(* Logix 5000 project; controller Close_Palletizing 1769-L33ERM rev 33.13; software revision 33.00; part 5 of 5 *)
(* tags used below, declared in another part *)
   ConveyorLocations_ONS : BOOL;
   Write_ActiveUserFrame2 : BOOL;
   ActiveUserFrame : DINT;
   ActiveUserFrame_Old : DINT;
   ActiveUserFrame_Timer : TIMER;
   ActiveUserFrameErr : BOOL;
   AirPressure : ALIAS FOR YRC1000_Rbt_Ctlr:I.Data[1].4;   // Sensor on air in, used to verify pressure
   BoltBucketSensor : ALIAS FOR YRC1000_Rbt_Ctlr:I.Data[1].7;   // Sense if the Bolt Bucket is present in the stand
   CenterDist : DINT;
   ConveyorApproachLocation : YRC1000_POSITION_VAR;
   ConveyorHeight : REAL;   // Distance from UF 3 to the top of the conveyor
   ConveyorPickLocation : YRC1000_POSITION_VAR;
   CurrentPos : REAL[6];   // Current position of the active TCP on the robot
   CurrentPos_micro : YRC1000_POSITION_VAR;   // μm
   currentPosErr : BOOL;
   CurrPos_Timer : TIMER;
   DoorRequestAccess : ALIAS FOR YRC1000_Rbt_Ctlr:I.Data[1].0;   // Door Interlock, For request Entry
   DoorUnlocked : ALIAS FOR YRC1000_Rbt_Ctlr:I.Data[2].0;   // The Door Latch is unlocked
   Error_RobotPickupFailed : ALIAS FOR YRC1000_Rbt_Ctlr:I.Data[9].3;
   GoToPartChange : ALIAS FOR YRC1000_Rbt_Ctlr:O.Data[6].0;
   HMI_Reset : BOOL;
   HMI_Stop : ALIAS FOR YRC1000_Rbt_Ctlr:O.Data[5].4;
   IFM_Port1_Stroke : Generic_4PORT_IOL;   // Stroke sensor reading can be found in StrokeInputArray[0]
   InPartChange : ALIAS FOR YRC1000_Rbt_Ctlr:I.Data[9].7;
   LayerNum : DINT;
   LeftPalletComplete : ALIAS FOR YRC1000_Rbt_Ctlr:O.Data[4].0;
   LeftPalletPresent : ALIAS FOR YRC1000_Rbt_Ctlr:O.Data[6].6;
   LeftPalletSensor : ALIAS FOR YRC1000_Rbt_Ctlr:I.Data[1].2;   // Sense if a pallet is in the pallet holder
   LeftPalletWillBeNew : BOOL;
   msg_Read_ActiveUserFrame : MESSAGE;
   msg_Read_CurrentPosition : MESSAGE;   // Reading the current position of the robot
   msg_Read_PalletCount : MESSAGE;
   msg_Read_PartCount : MESSAGE;   // Reading Part Count from the robot
   msg_Write_ActiveUserFrame : MESSAGE;
   msg_Write_ConveyorApproachLocation : MESSAGE;
   msg_Write_ConveyorPickLocation : MESSAGE;
   msg_Write_PalletCount : MESSAGE;
   msg_Write_PalletPlaceLocation : MESSAGE;
   msg_Write_PartCount : MESSAGE;
   msg_Write_RadiatorType : MESSAGE;
   OffsetDist : DINT;
   PalletCount : DINT;
   PalletCount_old : DINT;
   PalletCount_Timer : TIMER;
   PalletCountErr : BOOL;
   Palletizer_full_produced : DINT;
   PalletNotClear : ALIAS FOR YRC1000_Rbt_Ctlr:O.Data[6].5;
   PartCount : DINT;
   PartCount_Timer : TIMER;
   PartCountErr : BOOL;
   PartInTool : ALIAS FOR YRC1000_Rbt_Ctlr:O.Data[4].2;
   PartLength : DINT;
   PartLength_Current : DINT;   // 17" = 432 mm | 30" = 762 mm | 41" = 1041 mm
   PartNum : DINT;
   PartNum_Current : DINT;
   PartNumber : STRING;
   PartNumber_Current : STRING;
   PartPosition : DINT;
   PartRows : DINT;
   PartRows_Current : DINT;
   PartThickness : REAL;
   PartThickness_Current : REAL;   // 2r = 34.1-34.6 mm | 3r = 51.1-51.8 mm | 4r = 68.2-68.9 mm
   PartWidth : DINT;
   PartWidth_Current : DINT;   // 14" = 356 mm | 16" = 407 mm | 20" = 508 mm | 22" = 559 mm | 24" = 610 mm | 28" = 711 mm | 32" = 813 mm
   PickReq_State : DINT;
   PickRequest : ALIAS FOR YRC1000_Rbt_Ctlr:I.Data[9].6;
   PickRequestAcknowledge : ALIAS FOR YRC1000_Rbt_Ctlr:O.Data[5].5;
   PickupConveyorSensor : ALIAS FOR YRC1000_Rbt_Ctlr:I.Data[1].5;   // Sense if the radiator is ready for pickup
   Place_Error : BOOL;
   PlaceReq_State : DINT;
   PlaceRequestAcknowledge : ALIAS FOR YRC1000_Rbt_Ctlr:O.Data[4].5;
   PN_Timer : TIMER;
   QuadStack : ALIAS FOR YRC1000_Rbt_Ctlr:O.Data[5].1;
   RadiatorPlaceLocation : YRC1000_POSITION_VAR;
   RadiatorType : DINT;   // 1: 17" 2: 30" 3 41"
   Read_ActiveUserFrame : BOOL;
   Read_CurrPos : BOOL;
   Read_PalletCount : BOOL;
   Read_PartCount : BOOL;
   Reset : ALIAS FOR YRC1000_Rbt_Ctlr:I.Data[1].1;   // Door Interlock, For reset Entry
   ResetPalletCount : BOOL;
   RightPalletComplete : ALIAS FOR YRC1000_Rbt_Ctlr:O.Data[4].1;
   RightPalletPresent : ALIAS FOR YRC1000_Rbt_Ctlr:O.Data[6].7;
   RightPalletSensor : ALIAS FOR YRC1000_Rbt_Ctlr:I.Data[1].3;   // Sense if a pallet is in the pallet holder
   RightPalletWillBeNew : BOOL;
   RobotExternalEStop : ALIAS FOR YRC1000_Rbt_Ctlr:I.Data[4].1;
   RobotPlaceRequest : ALIAS FOR YRC1000_Rbt_Ctlr:I.Data[9].2;
   RobotTeachPendantEStop : ALIAS FOR YRC1000_Rbt_Ctlr:I.Data[4].2;
   Running : ALIAS FOR YRC1000_Rbt_Ctlr:I.Data[8].0;   // Robot running status
   SafetyCircuitBroken : ALIAS FOR YRC1000_Rbt_Ctlr:I.Data[4].0;
   SecondConveyorSensor : ALIAS FOR YRC1000_Rbt_Ctlr:I.Data[1].6;   // Sense if a coil is waiting on the conveyor
   SideDist : DINT;
   SingleStack : ALIAS FOR YRC1000_Rbt_Ctlr:O.Data[5].0;
   test_toggle : BOOL;
   ToolExtended : ALIAS FOR YRC1000_Rbt_Ctlr:O.Data[4].3;
   ToolRetracted : ALIAS FOR YRC1000_Rbt_Ctlr:O.Data[4].4;
   ToPC_AirPressure : DINT;
   ToPC_BoltBucketSensor : DINT;
   ToPC_ConveyorStatus : DINT;
   ToPC_DoorStatus : DINT;
   ToPC_FanucFault : DINT;
   ToPC_FanucRunning : DINT;
   ToPC_LeftPalletStatus : DINT;
   ToPC_PalletNotClear : DINT;
   ToPC_PickupFailed : DINT;
   ToPC_PlaceError : DINT;
   ToPC_RightPalletStatus : DINT;
   ToPC_RobotEStop : DINT;
   ToPC_RobotRunning : DINT;
   ToPC_SafetyCircuitBroken : DINT;
   ToPC_ToolStatus : DINT;
   TwoStack : ALIAS FOR YRC1000_Rbt_Ctlr:O.Data[6].2;
   WaitingForPartAtEnd : BOOL;
   Write_ActiveUserFrame : BOOL;
   Write_ActiveUserFrame1 : BOOL;
   Write_ConveyorLocations : BOOL;
   Write_PalletPlaceLocation : BOOL;
   Write_PartCount : BOOL;
   Write_RadiatorType : BOOL;
(* MainProgram, continued *)

ROUTINE Motoman_Messaging   (* ladder *)
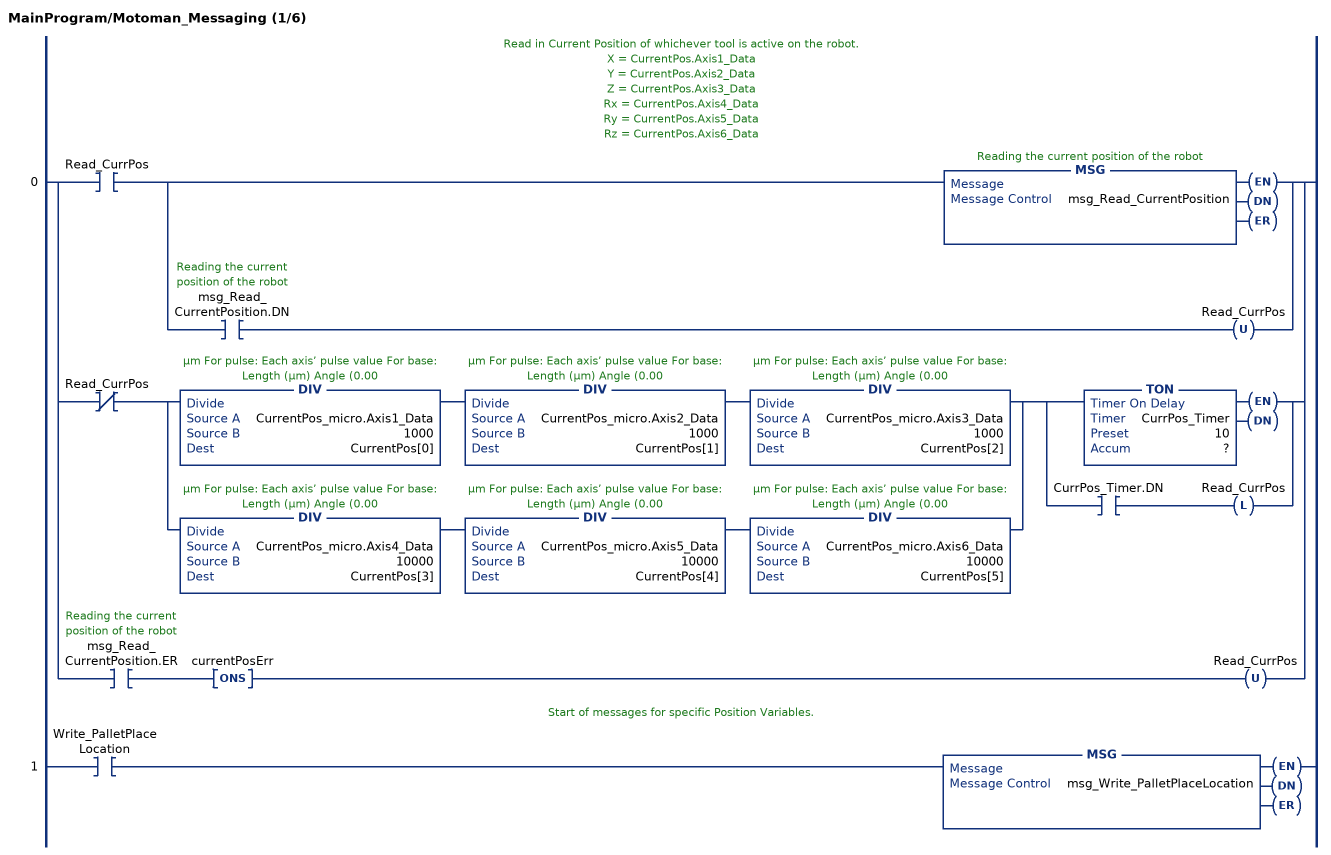
   // Read in Current Position of whichever tool is active on the robot.
   //  X = CurrentPos.Axis1_Data
   //  Y = CurrentPos.Axis2_Data
   //  Z = CurrentPos.Axis3_Data
   // Rx = CurrentPos.Axis4_Data
   // Ry = CurrentPos.Axis5_Data
   // Rz = CurrentPos.Axis6_Data
   0: [XIC(Read_CurrPos) [MSG(msg_Read_CurrentPosition) ,XIC(msg_Read_CurrentPosition.DN) OTU(Read_CurrPos) ] ,XIO(Read_CurrPos) [DIV(CurrentPos_micro.Axis1_Data,1000,CurrentPos[0]) DIV(CurrentPos_micro.Axis2_Data,1000,CurrentPos[1]) DIV(CurrentPos_micro.Axis3_Data,1000,CurrentPos[2]) ,DIV(CurrentPos_micro.Axis4_Data,10000,CurrentPos[3]) DIV(CurrentPos_micro.Axis5_Data,10000,CurrentPos[4]) DIV(CurrentPos_micro.Axis6_Data,10000,CurrentPos[5]) ] [TON(CurrPos_Timer,?,?) ,XIC(CurrPos_Timer.DN) OTL(Read_CurrPos) ] ,XIC(msg_Read_CurrentPosition.ER) ONS(currentPosErr) OTU(Read_CurrPos) ];
   // Start of messages for specific Position Variables.
   1: XIC(Write_PalletPlaceLocation)MSG(msg_Write_PalletPlaceLocation);
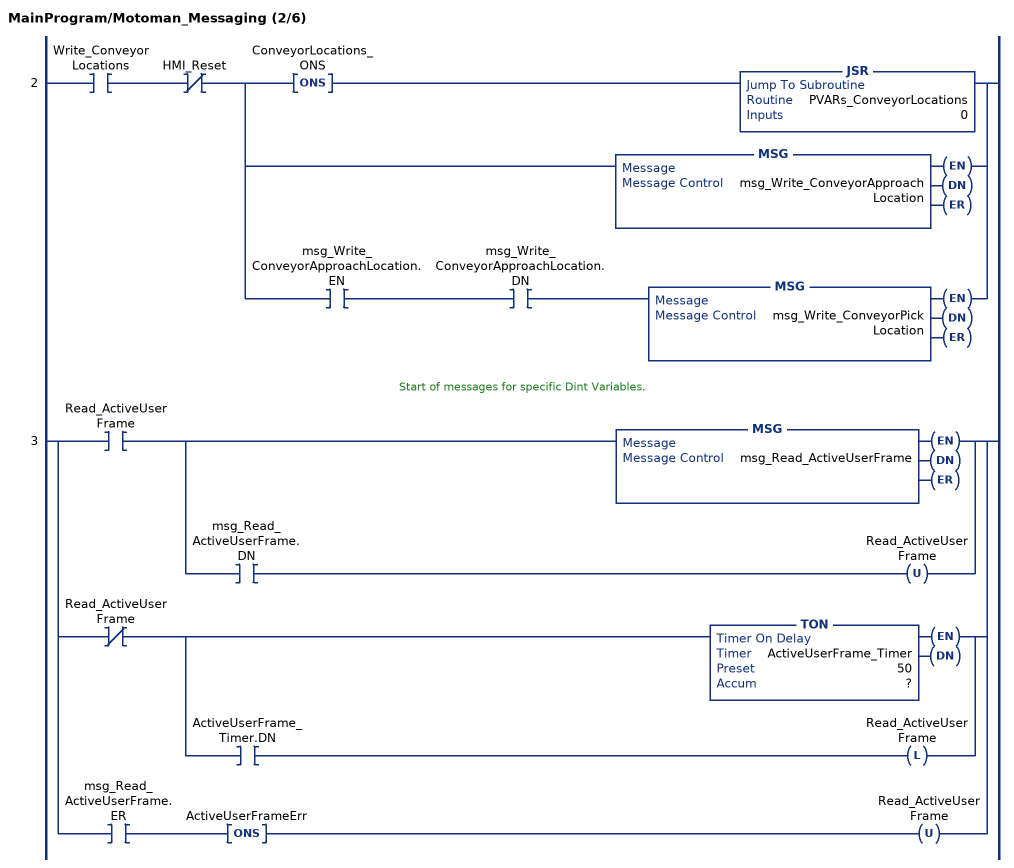
   2: XIC(Write_ConveyorLocations)XIO(HMI_Reset)[ONS(ConveyorLocations_ONS) JSR(PVARs_ConveyorLocations,0) ,MSG(msg_Write_ConveyorApproachLocation) ,XIC(msg_Write_ConveyorApproachLocation.EN) XIC(msg_Write_ConveyorApproachLocation.DN) MSG(msg_Write_ConveyorPickLocation) ];
   // Start of messages for specific Dint Variables.
   3: [XIC(Read_ActiveUserFrame) [MSG(msg_Read_ActiveUserFrame) ,XIC(msg_Read_ActiveUserFrame.DN) OTU(Read_ActiveUserFrame) ] ,XIO(Read_ActiveUserFrame) [TON(ActiveUserFrame_Timer,?,?) ,XIC(ActiveUserFrame_Timer.DN) OTL(Read_ActiveUserFrame) ] ,XIC(msg_Read_ActiveUserFrame.ER) ONS(ActiveUserFrameErr) OTU(Read_ActiveUserFrame) ];
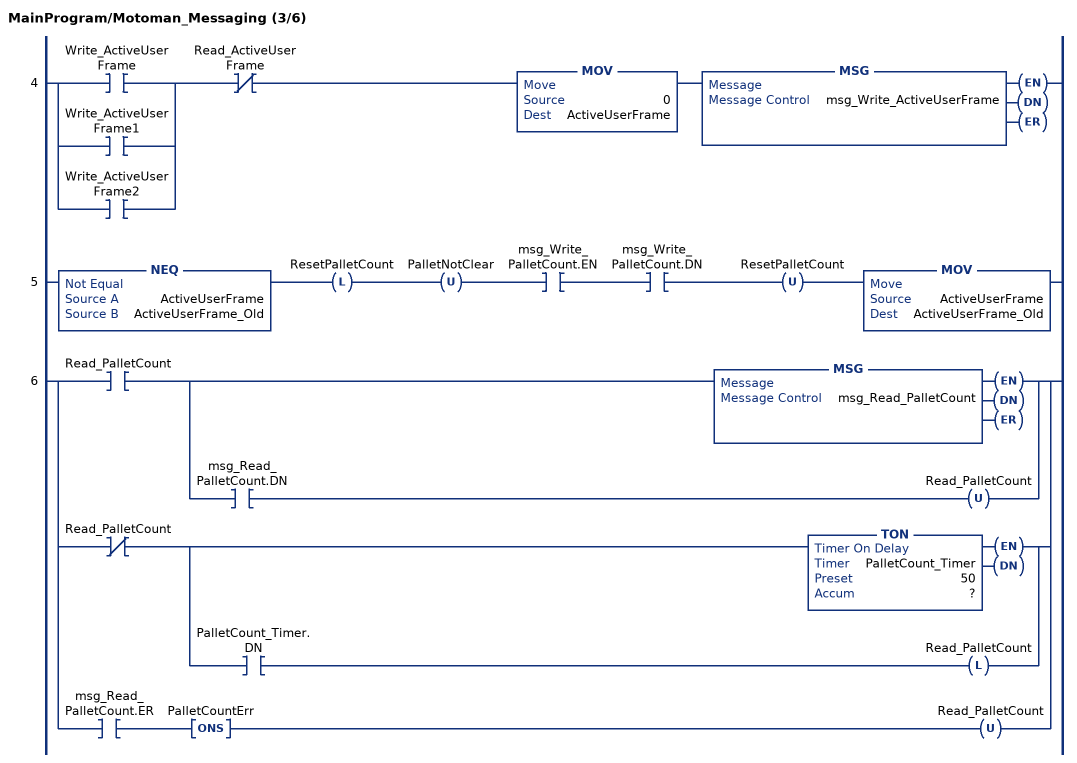
   4: [XIC(Write_ActiveUserFrame) ,XIC(Write_ActiveUserFrame1) ,XIC(Write_ActiveUserFrame2) ]XIO(Read_ActiveUserFrame)MOV(0,ActiveUserFrame)MSG(msg_Write_ActiveUserFrame);
   5: NEQ(ActiveUserFrame,ActiveUserFrame_Old)OTL(ResetPalletCount)OTU(PalletNotClear)XIC(msg_Write_PalletCount.EN)XIC(msg_Write_PalletCount.DN)OTU(ResetPalletCount)MOV(ActiveUserFrame,ActiveUserFrame_Old);
   6: [XIC(Read_PalletCount) [MSG(msg_Read_PalletCount) ,XIC(msg_Read_PalletCount.DN) OTU(Read_PalletCount) ] ,XIO(Read_PalletCount) [TON(PalletCount_Timer,?,?) ,XIC(PalletCount_Timer.DN) OTL(Read_PalletCount) ] ,XIC(msg_Read_PalletCount.ER) ONS(PalletCountErr) OTU(Read_PalletCount) ];
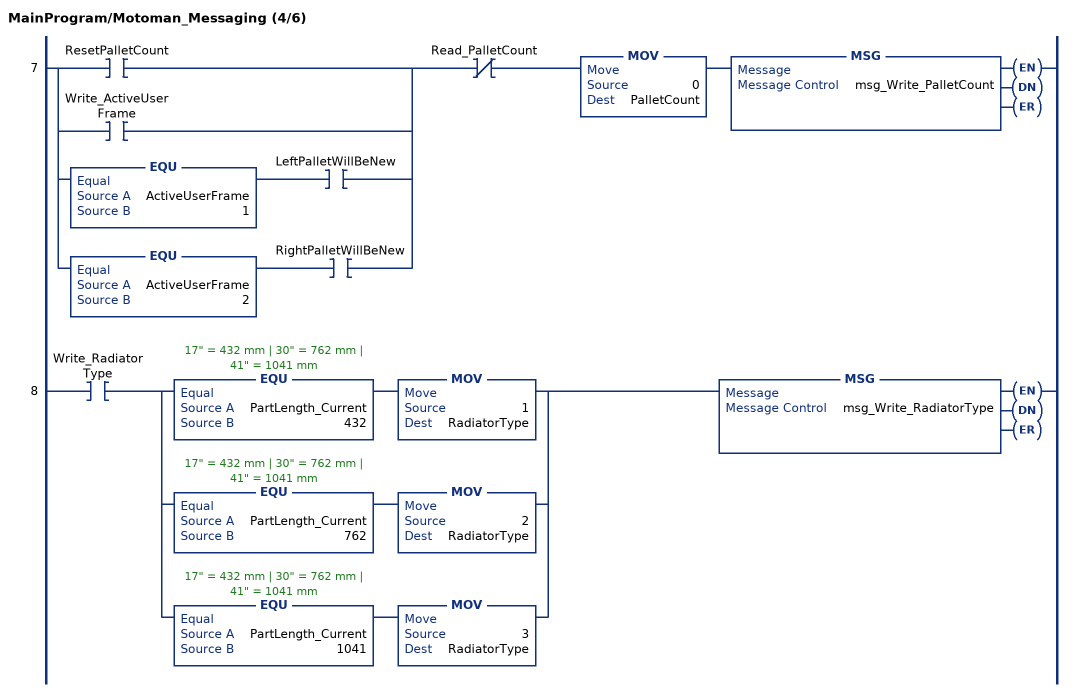
   7: [XIC(ResetPalletCount) ,XIC(Write_ActiveUserFrame) ,EQU(ActiveUserFrame,1) XIC(LeftPalletWillBeNew) ,EQU(ActiveUserFrame,2) XIC(RightPalletWillBeNew) ]XIO(Read_PalletCount)MOV(0,PalletCount)MSG(msg_Write_PalletCount);
   8: XIC(Write_RadiatorType)[EQU(PartLength_Current,432) MOV(1,RadiatorType) ,EQU(PartLength_Current,762) MOV(2,RadiatorType) ,EQU(PartLength_Current,1041) MOV(3,RadiatorType) ]MSG(msg_Write_RadiatorType);
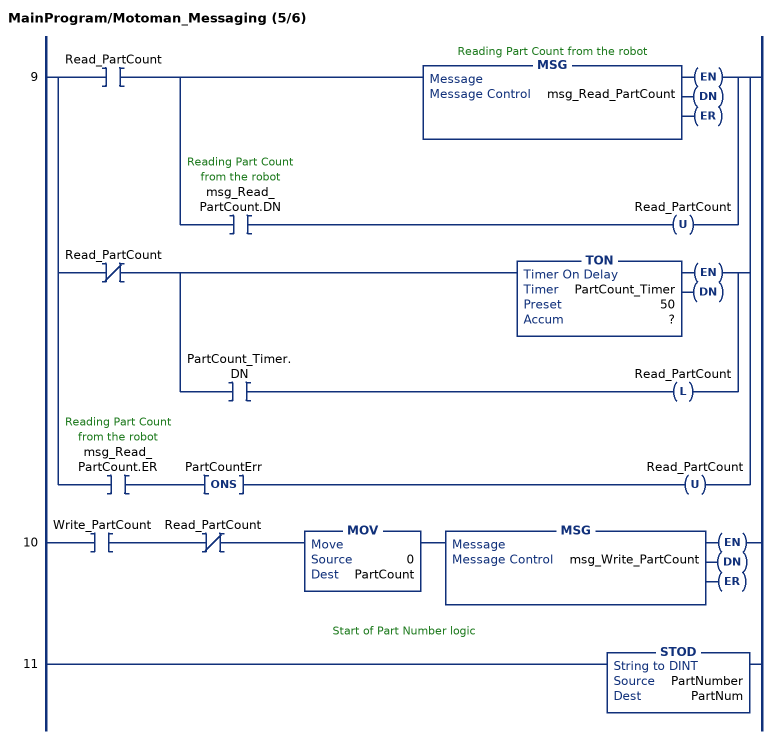
   9: [XIC(Read_PartCount) [MSG(msg_Read_PartCount) ,XIC(msg_Read_PartCount.DN) OTU(Read_PartCount) ] ,XIO(Read_PartCount) [TON(PartCount_Timer,?,?) ,XIC(PartCount_Timer.DN) OTL(Read_PartCount) ] ,XIC(msg_Read_PartCount.ER) ONS(PartCountErr) OTU(Read_PartCount) ];
   10: XIC(Write_PartCount)XIO(Read_PartCount)MOV(0,PartCount)MSG(msg_Write_PartCount);
   // Start of Part Number logic
   11: STOD(PartNumber,PartNum);
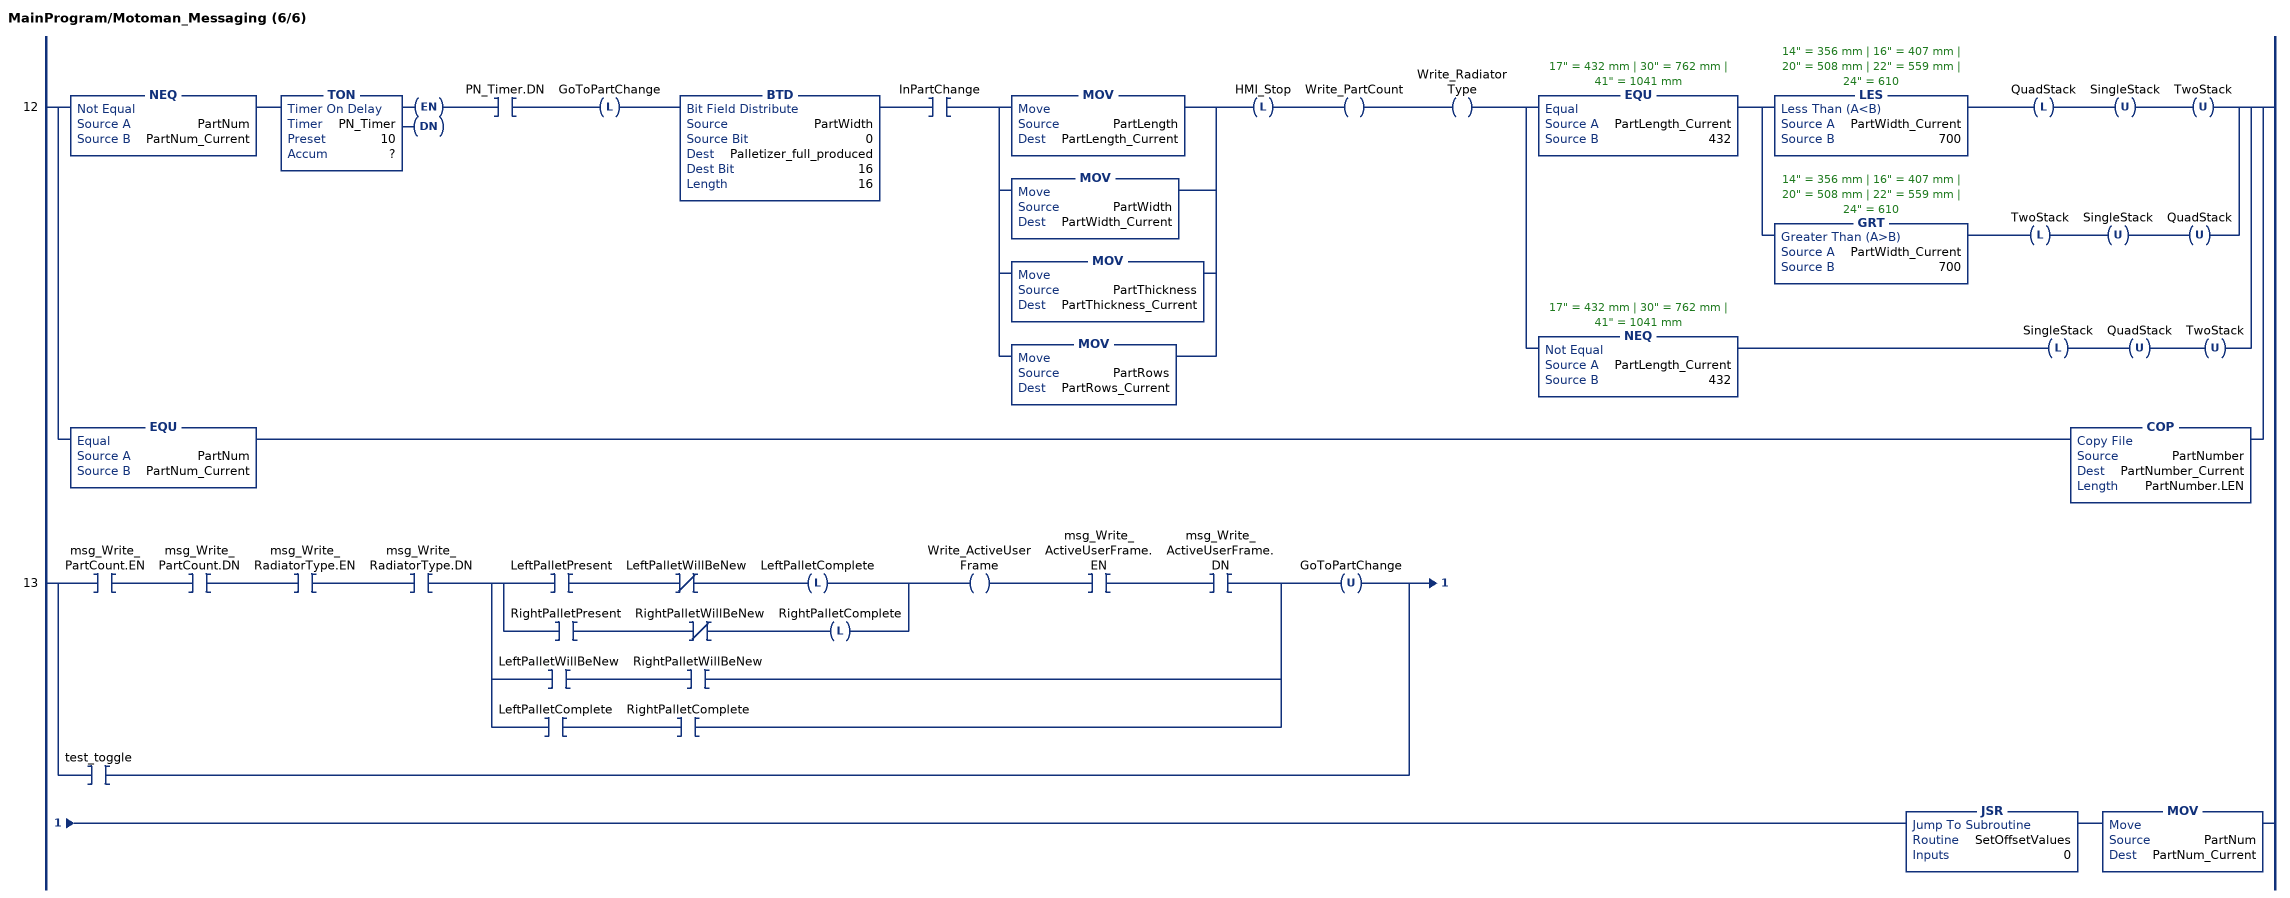
   12: [NEQ(PartNum,PartNum_Current) TON(PN_Timer,?,?) XIC(PN_Timer.DN) OTL(GoToPartChange) BTD(PartWidth,0,Palletizer_full_produced,16,16) XIC(InPartChange) [MOV(PartLength,PartLength_Current) ,MOV(PartWidth,PartWidth_Current) ,MOV(PartThickness,PartThickness_Current) ,MOV(PartRows,PartRows_Current) ] OTL(HMI_Stop) OTE(Write_PartCount) OTE(Write_RadiatorType) [EQU(PartLength_Current,432) [LES(PartWidth_Current,700) OTL(QuadStack) OTU(SingleStack) OTU(TwoStack) ,GRT(PartWidth_Current,700) OTL(TwoStack) OTU(SingleStack) OTU(QuadStack) ] ,NEQ(PartLength_Current,432) OTL(SingleStack) OTU(QuadStack) OTU(TwoStack) ] ,EQU(PartNum,PartNum_Current) COP(PartNumber,PartNumber_Current,PartNumber.LEN) ];
   13: [XIC(msg_Write_PartCount.EN) XIC(msg_Write_PartCount.DN) XIC(msg_Write_RadiatorType.EN) XIC(msg_Write_RadiatorType.DN) [[XIC(LeftPalletPresent) XIO(LeftPalletWillBeNew) OTL(LeftPalletComplete) ,XIC(RightPalletPresent) XIO(RightPalletWillBeNew) OTL(RightPalletComplete) ] OTE(Write_ActiveUserFrame) XIC(msg_Write_ActiveUserFrame.EN) XIC(msg_Write_ActiveUserFrame.DN) ,[XIC(LeftPalletWillBeNew) XIC(RightPalletWillBeNew) ,XIC(LeftPalletComplete) XIC(RightPalletComplete) ] ] OTU(GoToPartChange) ,XIC(test_toggle) ]JSR(SetOffsetValues,0)MOV(PartNum,PartNum_Current);
END_ROUTINE

ROUTINE PC_TagVariables   (* ladder *)
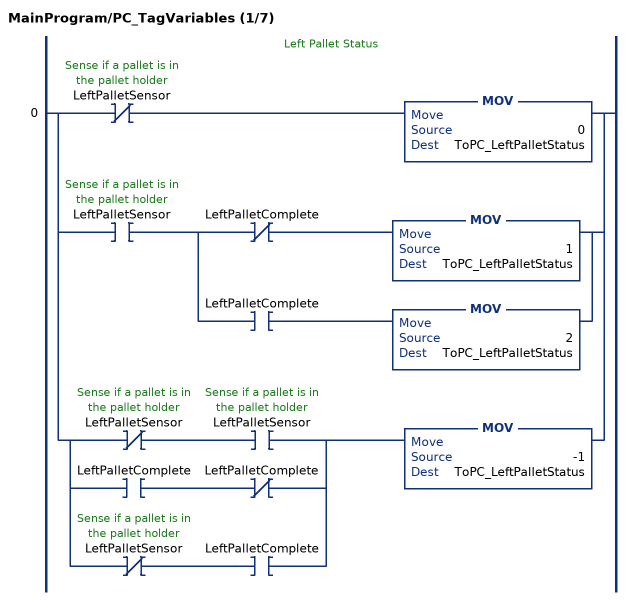
   // Left Pallet Status
   0: [[XIO(LeftPalletSensor) MOV(0,ToPC_LeftPalletStatus) ,XIC(LeftPalletSensor) [XIO(LeftPalletComplete) MOV(1,ToPC_LeftPalletStatus) ,XIC(LeftPalletComplete) MOV(2,ToPC_LeftPalletStatus) ] ] ,[XIO(LeftPalletSensor) XIC(LeftPalletSensor) ,XIC(LeftPalletComplete) XIO(LeftPalletComplete) ,XIO(LeftPalletSensor) XIC(LeftPalletComplete) ] MOV(-1,ToPC_LeftPalletStatus) ];
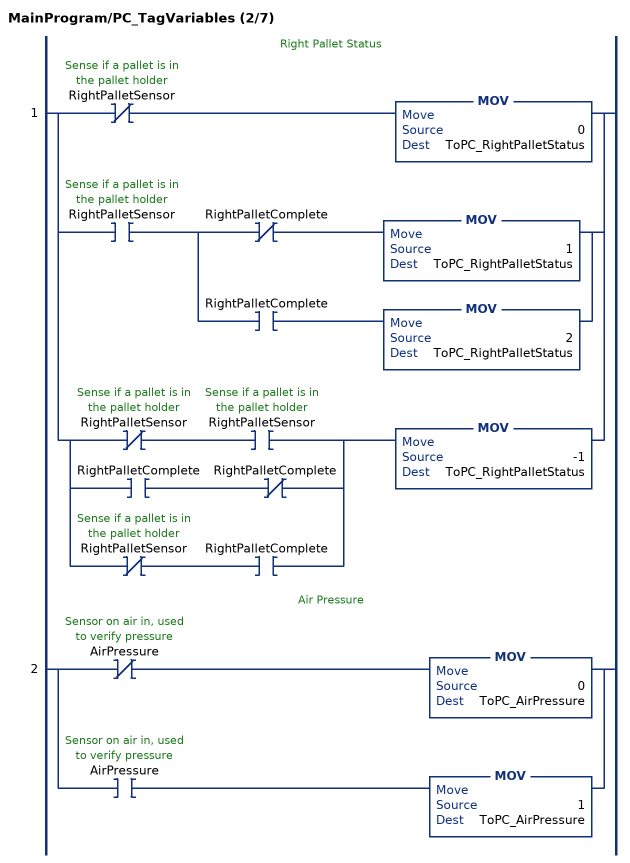
   // Right Pallet Status
   1: [[XIO(RightPalletSensor) MOV(0,ToPC_RightPalletStatus) ,XIC(RightPalletSensor) [XIO(RightPalletComplete) MOV(1,ToPC_RightPalletStatus) ,XIC(RightPalletComplete) MOV(2,ToPC_RightPalletStatus) ] ] ,[XIO(RightPalletSensor) XIC(RightPalletSensor) ,XIC(RightPalletComplete) XIO(RightPalletComplete) ,XIO(RightPalletSensor) XIC(RightPalletComplete) ] MOV(-1,ToPC_RightPalletStatus) ];
   // Air Pressure
   2: [XIO(AirPressure) MOV(0,ToPC_AirPressure) ,XIC(AirPressure) MOV(1,ToPC_AirPressure) ];
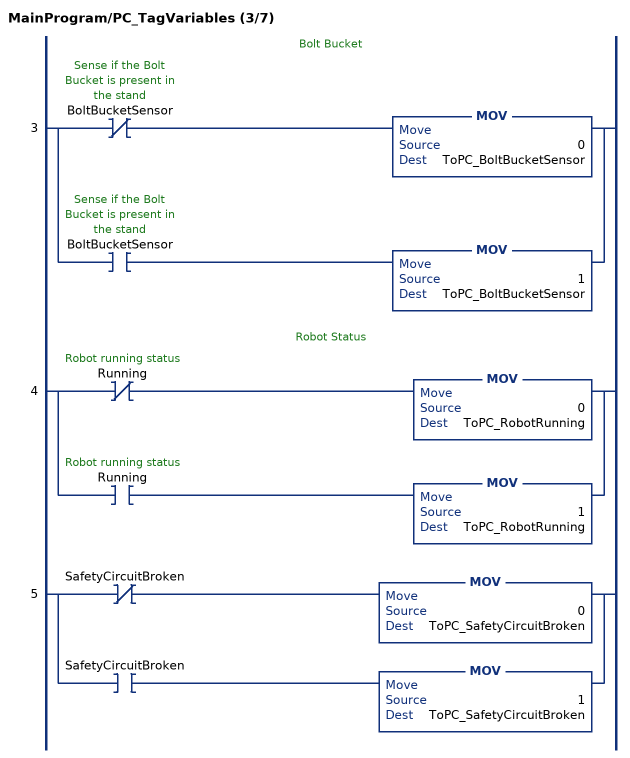
   // Bolt Bucket
   3: [XIO(BoltBucketSensor) MOV(0,ToPC_BoltBucketSensor) ,XIC(BoltBucketSensor) MOV(1,ToPC_BoltBucketSensor) ];
   // Robot Status
   4: [XIO(Running) MOV(0,ToPC_RobotRunning) ,XIC(Running) MOV(1,ToPC_RobotRunning) ];
   5: [XIO(SafetyCircuitBroken) MOV(0,ToPC_SafetyCircuitBroken) ,XIC(SafetyCircuitBroken) MOV(1,ToPC_SafetyCircuitBroken) ];
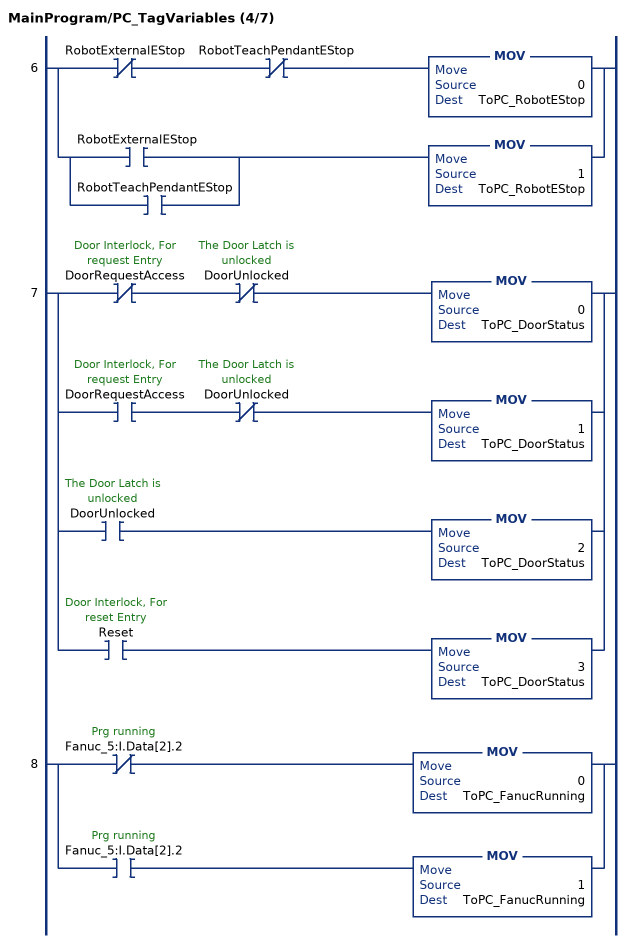
   6: [XIO(RobotExternalEStop) XIO(RobotTeachPendantEStop) MOV(0,ToPC_RobotEStop) ,[XIC(RobotExternalEStop) ,XIC(RobotTeachPendantEStop) ] MOV(1,ToPC_RobotEStop) ];
   7: [XIO(DoorRequestAccess) XIO(DoorUnlocked) MOV(0,ToPC_DoorStatus) ,XIC(DoorRequestAccess) XIO(DoorUnlocked) MOV(1,ToPC_DoorStatus) ,XIC(DoorUnlocked) MOV(2,ToPC_DoorStatus) ,XIC(Reset) MOV(3,ToPC_DoorStatus) ];
   8: [XIO(Fanuc_5:I.Data[2].2) MOV(0,ToPC_FanucRunning) ,XIC(Fanuc_5:I.Data[2].2) MOV(1,ToPC_FanucRunning) ];
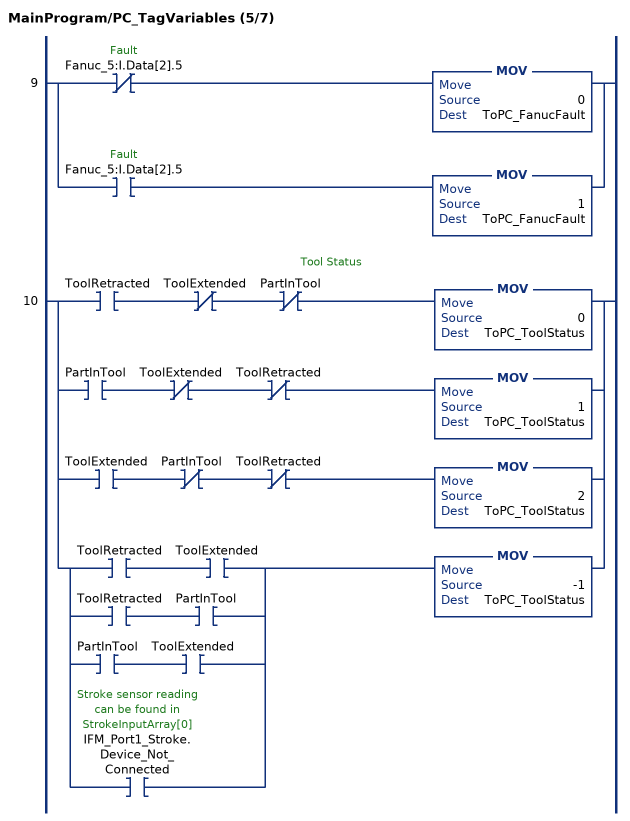
   9: [XIO(Fanuc_5:I.Data[2].5) MOV(0,ToPC_FanucFault) ,XIC(Fanuc_5:I.Data[2].5) MOV(1,ToPC_FanucFault) ];
   // Tool Status
   10: [XIC(ToolRetracted) XIO(ToolExtended) XIO(PartInTool) MOV(0,ToPC_ToolStatus) ,XIC(PartInTool) XIO(ToolExtended) XIO(ToolRetracted) MOV(1,ToPC_ToolStatus) ,XIC(ToolExtended) XIO(PartInTool) XIO(ToolRetracted) MOV(2,ToPC_ToolStatus) ,[XIC(ToolRetracted) XIC(ToolExtended) ,XIC(ToolRetracted) XIC(PartInTool) ,XIC(PartInTool) XIC(ToolExtended) ,XIC(IFM_Port1_Stroke.Device_Not_Connected) ] MOV(-1,ToPC_ToolStatus) ];
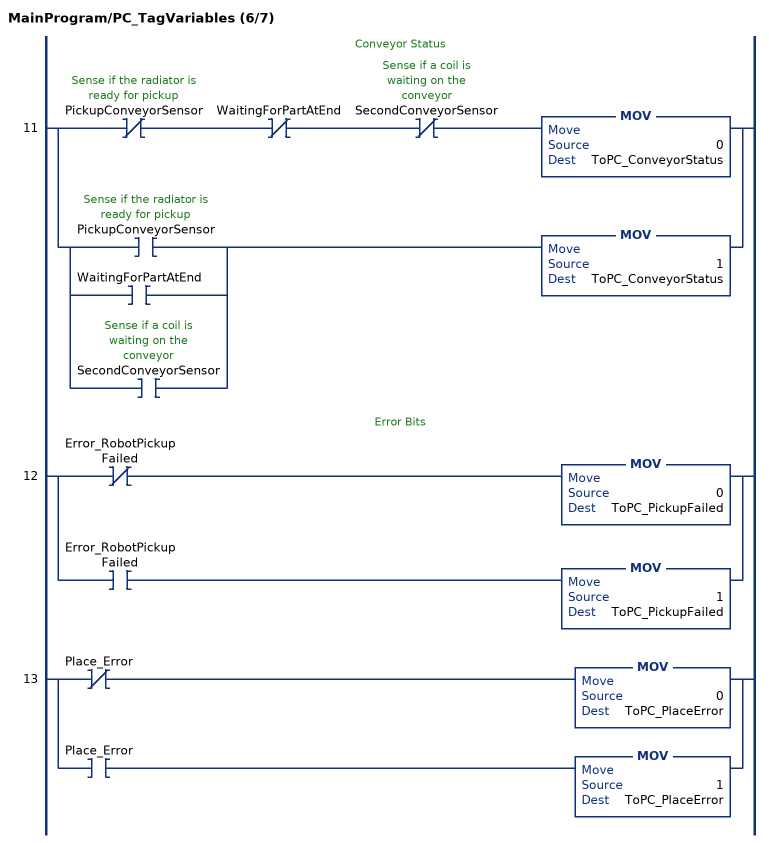
   // Conveyor Status
   11: [XIO(PickupConveyorSensor) XIO(WaitingForPartAtEnd) XIO(SecondConveyorSensor) MOV(0,ToPC_ConveyorStatus) ,[XIC(PickupConveyorSensor) ,XIC(WaitingForPartAtEnd) ,XIC(SecondConveyorSensor) ] MOV(1,ToPC_ConveyorStatus) ];
   // Error Bits
   12: [XIO(Error_RobotPickupFailed) MOV(0,ToPC_PickupFailed) ,XIC(Error_RobotPickupFailed) MOV(1,ToPC_PickupFailed) ];
   13: [XIO(Place_Error) MOV(0,ToPC_PlaceError) ,XIC(Place_Error) MOV(1,ToPC_PlaceError) ];
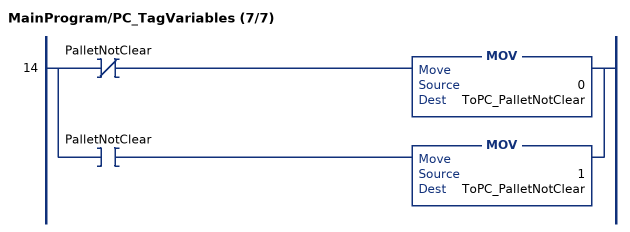
   14: [XIO(PalletNotClear) MOV(0,ToPC_PalletNotClear) ,XIC(PalletNotClear) MOV(1,ToPC_PalletNotClear) ];
END_ROUTINE

ROUTINE PVARs_ConveyorLocations   (* structured text *)
   // Set tool number and Ry based on PartLength
   if PartLength_Current = 432 then
   	ConveyorApproachLocation.Tool_Num := 2;
   	ConveyorApproachLocation.Axis5_Data := 20000;
   
   	ConveyorPickLocation.Tool_Num := 2;
   	ConveyorPickLocation.Axis5_Data := 20000;
   elsif PartLength_Current = 762 then
   	ConveyorApproachLocation.Tool_Num := 3;
   	ConveyorApproachLocation.Axis5_Data := 15000;
   
   	ConveyorPickLocation.Tool_Num := 3;
   	ConveyorPickLocation.Axis5_Data := 15000;
   elsif PartLength_Current = 1041 then
   	ConveyorApproachLocation.Tool_Num := 4;
   	ConveyorApproachLocation.Axis5_Data := 10000;
   
   	ConveyorPickLocation.Tool_Num := 4;
   	ConveyorPickLocation.Axis5_Data := 10000;
   end_if;
   
   // Set X value based on conveyor height and part dimensions
   ConveyorPickLocation.Axis1_Data := (ConveyorHeight - PartLength_Current) * 1000;
   if PartLength_Current = 432 then
   	ConveyorPickLocation.Axis1_Data := ConveyorPickLocation.Axis1_Data - 20000;
   elsif PartLength_Current = 762 then
   	ConveyorPickLocation.Axis1_Data := ConveyorPickLocation.Axis1_Data - 14000;
   elsif PartLength_Current = 1041 then
   	ConveyorPickLocation.Axis1_Data := ConveyorPickLocation.Axis1_Data - 14000;
   end_if;
   ConveyorApproachLocation.Axis1_Data := ConveyorPickLocation.Axis1_Data;
   
   // Set Y value of ConveyorPickLocation based on PartWidth
   ConveyorPickLocation.Axis2_Data := (PartWidth_Current / 2) * 1000;
   if ConveyorPickLocation.Axis2_Data > 360000 then
   	ConveyorPickLocation.Axis2_Data := 360000;
   	SideDist := ((PartWidth_Current / 2) * 1000) - 360000;
   else
   	SideDist := 0;
   end_if;
   
   // Set Z value of ConveyorPickLocation based on PartThickness
   ConveyorPickLocation.Axis3_Data := (PartThickness_Current + 30) * 1000;
END_ROUTINE

ROUTINE PVARs_PlacePosition_QuadStack   (* structured text *)
   // This routine sets the variable data for the radiator placement position based on the pre-defined Offset values.
   
   // This is constant
   RadiatorPlaceLocation.Tool_Num := 8;
   
   LayerNum := (PalletCount / 4) + 1;
   PartPosition := PalletCount MOD 8;
   
   // Set X, Y, and Rz based on which position the radiator is being placed at
   if PartPosition = 0 then
   	RadiatorPlaceLocation.Axis1_Data := CenterDist + OffsetDist;
   	RadiatorPlaceLocation.Axis2_Data := CenterDist + SideDist;
   	RadiatorPlaceLocation.Axis6_Data := 0;
   elsif PartPosition = 1 then
   	RadiatorPlaceLocation.Axis1_Data := -CenterDist - SideDist;
   	RadiatorPlaceLocation.Axis2_Data := CenterDist + OffsetDist;
   	RadiatorPlaceLocation.Axis6_Data := 900000;
   elsif PartPosition = 2 then
   	RadiatorPlaceLocation.Axis1_Data := -CenterDist - OffsetDist;
   	RadiatorPlaceLocation.Axis2_Data := -CenterDist - SideDist;
   	RadiatorPlaceLocation.Axis6_Data := 1800000;
   elsif PartPosition = 3 then
   	RadiatorPlaceLocation.Axis1_Data := CenterDist + SideDist;
   	RadiatorPlaceLocation.Axis2_Data := -CenterDist - OffsetDist;
   	RadiatorPlaceLocation.Axis6_Data := -900000;
   elsif PartPosition = 4 then
   	RadiatorPlaceLocation.Axis1_Data := CenterDist + OffsetDist;
   	RadiatorPlaceLocation.Axis2_Data := -CenterDist + SideDist;
   	RadiatorPlaceLocation.Axis6_Data := 0;
   elsif PartPosition = 5 then
   	RadiatorPlaceLocation.Axis1_Data := CenterDist - SideDist;
   	RadiatorPlaceLocation.Axis2_Data := CenterDist + OffsetDist;
   	RadiatorPlaceLocation.Axis6_Data := 900000;
   elsif PartPosition = 6 then
   	RadiatorPlaceLocation.Axis1_Data := -CenterDist - OffsetDist;
   	RadiatorPlaceLocation.Axis2_Data := CenterDist - SideDist;
   	RadiatorPlaceLocation.Axis6_Data := 1800000;
   elsif PartPosition = 7 then
   	RadiatorPlaceLocation.Axis1_Data := -CenterDist + SideDist;
   	RadiatorPlaceLocation.Axis2_Data := -CenterDist - OffsetDist;
   	RadiatorPlaceLocation.Axis6_Data := -900000;
   end_if;
   
   // Account for all PartThickness plus the topmost and bottommost brackets
   	// Additional 100 mm up so we don't hit other radiators on our way to the location
   RadiatorPlaceLocation.Axis3_Data := ((LayerNum * PartThickness_Current) + 11.25 + 100 + 4) * 1000;
   if PartWidth_Current > 500 and PartWidth_Current < 600 then
   	// Radiators that are 20" or 22" wide have brackets resting on fins, so account for half of the internal brackets
   	RadiatorPlaceLocation.Axis3_Data := RadiatorPlaceLocation.Axis3_Data + ((LayerNum - 1) * 11.25) * 1000;
   elsif PartWidth_Current > 600 then
   	// Radiators that are 24+" wide have brackets resting on brackets, so account for all internal brackets
   	RadiatorPlaceLocation.Axis3_Data := RadiatorPlaceLocation.Axis3_Data + ((LayerNum - 1) * 22.5) * 1000;
   end_if;
END_ROUTINE

ROUTINE PVARs_PlacePosition_SingleStack   (* structured text *)
   /*
   	This routine sets the variable data for the radiator placement position.
   
   	The center of every radiator will be 0,0 in the user frame, so the only offset we need is:
   		OffsetDist = PartHeight / 2
   */
   
   // ToolNum depends on the part height
   if PartLength_Current = 762 then
   	RadiatorPlaceLocation.Tool_Num := 9;
   elsif PartLength_Current = 1041 then
   	RadiatorPlaceLocation.Tool_Num := 10;
   end_if;
   
   // Set LayerNum
   LayerNum := PalletCount + 1;
   
   if LayerNum MOD 2 = 1 then
   	RadiatorPlaceLocation.Axis1_Data := OffsetDist;
   	RadiatorPlaceLocation.Axis2_Data := SideDist;
   	RadiatorPlaceLocation.Axis6_Data := 0;
   else
   	if ActiveUserFrame = 1 then
   		RadiatorPlaceLocation.Axis1_Data := SideDist;
   		RadiatorPlaceLocation.Axis2_Data := -OffsetDist;
   		RadiatorPlaceLocation.Axis6_Data := -900000;
   	elsif ActiveUserFrame = 2 then
   		RadiatorPlaceLocation.Axis1_Data := -SideDist;
   		RadiatorPlaceLocation.Axis2_Data := OffsetDist;
   		RadiatorPlaceLocation.Axis6_Data := 900000;
   	end_if;
   end_if;
   
   // Set Z based on Part Thickness and the current layer number
   RadiatorPlaceLocation.Axis3_Data := ((LayerNum * PartThickness_Current) + 11.25 + 100 + 6) * 1000;
END_ROUTINE

ROUTINE PVARs_PlacePosition_TwoStack   (* structured text *)
   // This is constant
   RadiatorPlaceLocation.Tool_Num := 8;
   
   LayerNum := (PalletCount / 2) + 1;
   PartPosition := PalletCount MOD 4;
   
   // Set X, Y, and Rz based on which position the radiator is being placed at
   if PartPosition = 0 then
   	RadiatorPlaceLocation.Axis1_Data := CenterDist + OffsetDist;
   	RadiatorPlaceLocation.Axis2_Data := SideDist;
   	RadiatorPlaceLocation.Axis6_Data := 0;
   elsif PartPosition = 1 then
   	if ActiveUserFrame = 1 then
   		RadiatorPlaceLocation.Axis1_Data := -CenterDist + SideDist;
   		RadiatorPlaceLocation.Axis2_Data := -OffsetDist;
   		RadiatorPlaceLocation.Axis6_Data := -900000;
   	elsif ActiveUserFrame = 2 then
   		RadiatorPlaceLocation.Axis1_Data := -CenterDist - SideDist;
   		RadiatorPlaceLocation.Axis2_Data := OffsetDist;
   		RadiatorPlaceLocation.Axis6_Data := 900000;
   	end_if;
   elsif PartPosition = 2 then
   	RadiatorPlaceLocation.Axis1_Data := -CenterDist - OffsetDist;
   	RadiatorPlaceLocation.Axis2_Data := -SideDist;
   	RadiatorPlaceLocation.Axis6_Data := 1800000;
   elsif PartPosition = 3 then
   	if ActiveUserFrame = 1 then
   		RadiatorPlaceLocation.Axis1_Data := CenterDist + SideDist;
   		RadiatorPlaceLocation.Axis2_Data := -OffsetDist;
   		RadiatorPlaceLocation.Axis6_Data := -900000;
   	elsif ActiveUserFrame = 2 then
   		RadiatorPlaceLocation.Axis1_Data := CenterDist - SideDist;
   		RadiatorPlaceLocation.Axis2_Data := OffsetDist;
   		RadiatorPlaceLocation.Axis6_Data := 900000;
   	end_if;
   end_if;
   
   // Set Z based on Part Thickness and current layer number
   RadiatorPlaceLocation.Axis3_Data := ((LayerNum * PartThickness_Current) + 11.25 + ((LayerNum - 1) * 22.5) + 100 + 6) * 1000;
END_ROUTINE

ROUTINE Request_Pick   (* ladder *)
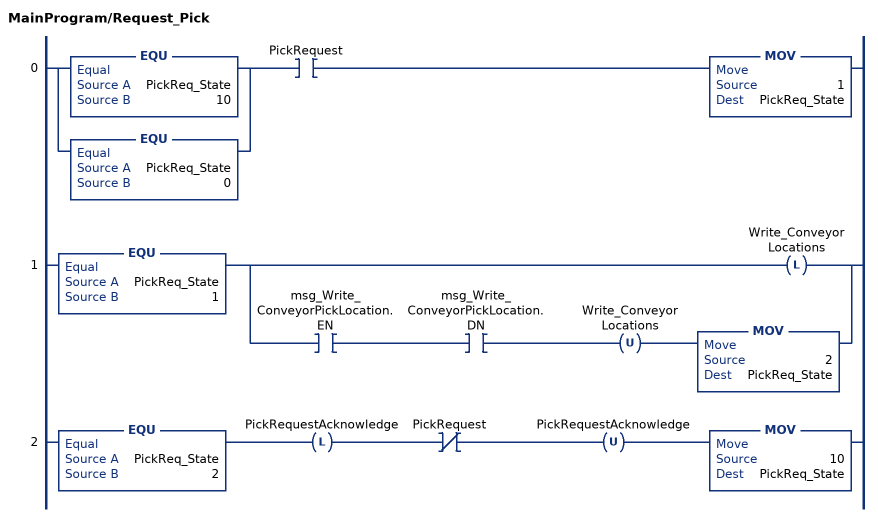
   0: [EQU(PickReq_State,10) ,EQU(PickReq_State,0) ]XIC(PickRequest)MOV(1,PickReq_State);
   1: EQU(PickReq_State,1)[OTL(Write_ConveyorLocations) ,XIC(msg_Write_ConveyorPickLocation.EN) XIC(msg_Write_ConveyorPickLocation.DN) OTU(Write_ConveyorLocations) MOV(2,PickReq_State) ];
   2: EQU(PickReq_State,2)OTL(PickRequestAcknowledge)XIO(PickRequest)OTU(PickRequestAcknowledge)MOV(10,PickReq_State);
END_ROUTINE

ROUTINE Request_Place   (* ladder *)
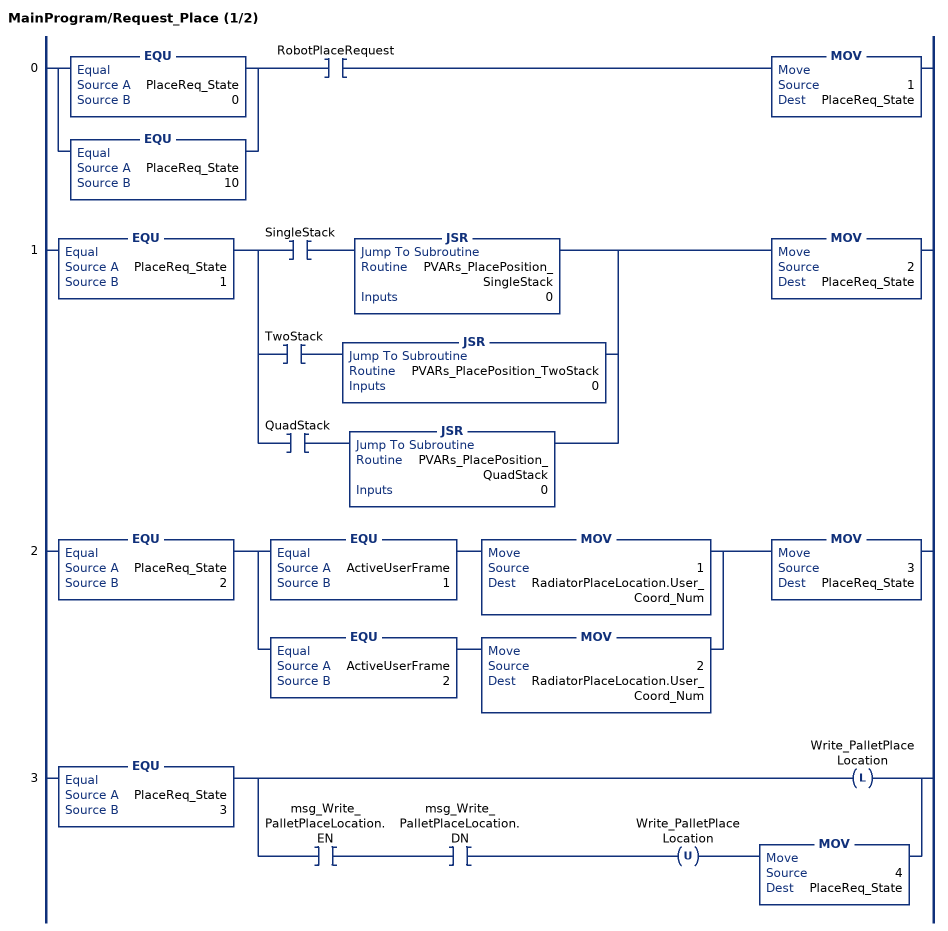
   0: [EQU(PlaceReq_State,0) ,EQU(PlaceReq_State,10) ]XIC(RobotPlaceRequest)MOV(1,PlaceReq_State);
   1: EQU(PlaceReq_State,1)[XIC(SingleStack) JSR(PVARs_PlacePosition_SingleStack,0) ,XIC(TwoStack) JSR(PVARs_PlacePosition_TwoStack,0) ,XIC(QuadStack) JSR(PVARs_PlacePosition_QuadStack,0) ]MOV(2,PlaceReq_State);
   2: EQU(PlaceReq_State,2)[EQU(ActiveUserFrame,1) MOV(1,RadiatorPlaceLocation.User_Coord_Num) ,EQU(ActiveUserFrame,2) MOV(2,RadiatorPlaceLocation.User_Coord_Num) ]MOV(3,PlaceReq_State);
   3: EQU(PlaceReq_State,3)[OTL(Write_PalletPlaceLocation) ,XIC(msg_Write_PalletPlaceLocation.EN) XIC(msg_Write_PalletPlaceLocation.DN) OTU(Write_PalletPlaceLocation) MOV(4,PlaceReq_State) ];
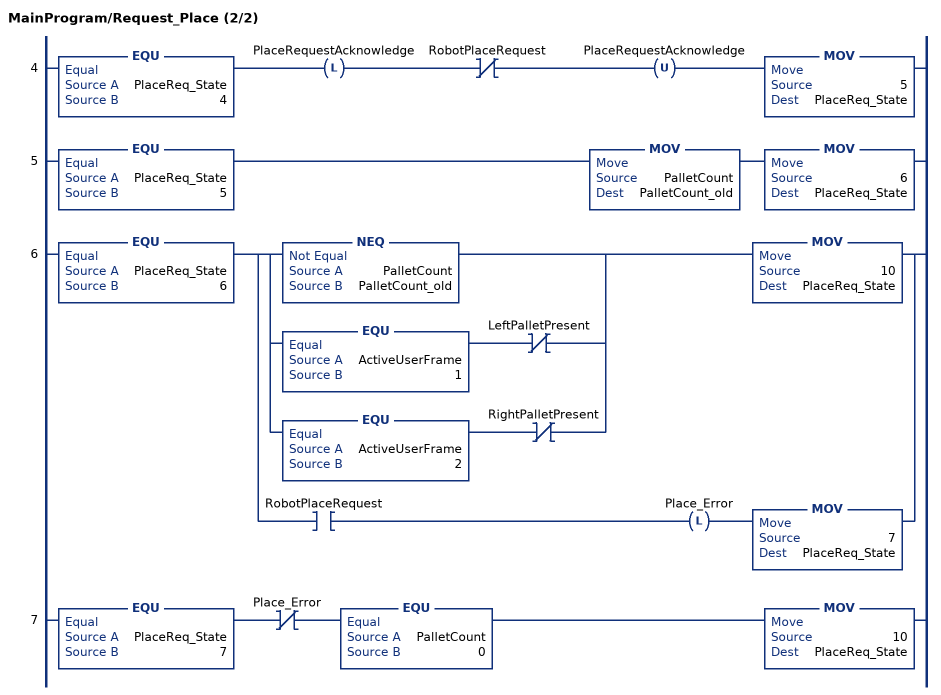
   4: EQU(PlaceReq_State,4)OTL(PlaceRequestAcknowledge)XIO(RobotPlaceRequest)OTU(PlaceRequestAcknowledge)MOV(5,PlaceReq_State);
   5: EQU(PlaceReq_State,5)MOV(PalletCount,PalletCount_old)MOV(6,PlaceReq_State);
   6: EQU(PlaceReq_State,6)[[NEQ(PalletCount,PalletCount_old) ,EQU(ActiveUserFrame,1) XIO(LeftPalletPresent) ,EQU(ActiveUserFrame,2) XIO(RightPalletPresent) ] MOV(10,PlaceReq_State) ,XIC(RobotPlaceRequest) OTL(Place_Error) MOV(7,PlaceReq_State) ];
   7: EQU(PlaceReq_State,7)XIO(Place_Error)EQU(PalletCount,0)MOV(10,PlaceReq_State);
END_ROUTINE

ROUTINE SetOffsetValues   (* structured text *)
   /*
   	CenterDist and OffsetDist are set when the part number changes.
   	These are based on part dimensions and stack pattern.
   */
   
   if PartLength_Current = 432 then
   	if PartWidth_Current > 700 then
   		CenterDist := (((PartLength_Current/2 + PartWidth_Current/2 + 35) / 2)) * 1000;
   	else
   		if PartWidth_Current > PartLength_Current then
   			CenterDist := (((PartLength_Current/2 + PartWidth_Current/2 + 35) / 2)) * 1000;
   		else
   			CenterDist := (((PartLength_Current/2 + PartLength_Current/2 + 35) / 2)) * 1000;
   		end_if;
   	end_if;
   else
   	CenterDist := 0;
   end_if;
   
   OffsetDist := ((PartLength_Current / 2) - 2) * 1000;
END_ROUTINE
END_PROGRAM
